// TwinCAT 3 PLC project Test
// ProgramVersion: 3.1.4024.0
// libraries:
//   Tc2_EtherCAT, * (Beckhoff Automation GmbH)
//   Tc2_Standard, * (Beckhoff Automation GmbH)
//   Tc2_System, * (Beckhoff Automation GmbH)
//   Tc3_Module, * (Beckhoff Automation GmbH)
// project tree:
//   DUTs/STRUCT/ Meca500SmPdo.TcDUT, SensorSmPdo.TcDUT
//   GVLs/ GVL.TcGVL
//   / PlcTask.TcTTO
//   POUs/ MAIN.TcPOU, Overall.TcPOU
// real-time tasks:
//   TASK PlcTask: cycle T#10ms, priority 20, ADS port 350
// I/O:
//   DEVICE Device 1 (EtherCAT), AmsNetId 192.168.0.153.2.1
//     Box 1 (Meca500) [Meca500]
//     Box 2 (Meca500) [Meca500]
//     Box 3 (BFT-MEDS-ECAT-M8) [BFT]
// variable links:
//   Test/Test Instance <-> Device 1 (EtherCAT)/Box 1 (Meca500)
//     PlcTask Inputs/GVL.Robot1.Inputs <-> SmPdoVariables/Meca500_SM_3
//     PlcTask Outputs/GVL.Robot1.Outputs <-> SmPdoVariables/Meca500_SM_2
//   Test/Test Instance <-> Device 1 (EtherCAT)/Box 2 (Meca500)
//     PlcTask Inputs/GVL.Robot2.Inputs <-> SmPdoVariables/Meca500_SM_3
//     PlcTask Outputs/GVL.Robot2.Outputs <-> SmPdoVariables/Meca500_SM_2
//   Test/Test Instance <-> Device 1 (EtherCAT)/Box 3 (BFT-MEDS-ECAT-M8)
//     PlcTask Inputs/GVL.Sensor.Inputs <-> SmPdoVariables/BFT_SM_3

CONFIGURATION Test
    RESOURCE PLC ON TwinCAT3
        TASK PlcTask(INTERVAL := T#10ms, PRIORITY := 20);
        PROGRAM MAIN WITH PlcTask : MAIN;
    END_RESOURCE
END_CONFIGURATION

// ---- DUTs/STRUCT/Meca500SmPdo.TcDUT
TYPE Meca500SmPdo :
STRUCT
	//From Ethercat Device SmPdos, Create this Structure by Enabling Create Sm/Pdo variable , in the Ethercat tab/Advance/Behavior
	Inputs 	AT %I* : ECAT_Meca500_SM_34A3A44A;	//for specific ESI firmware
	Outputs AT %Q* : ECAT_Meca500_SM_A587449F;	//for specific ESI firmware
	
	Connect					:	BOOL;	//Switch between Init State & OP State
	Connected				:	BOOL;	//Validate OP State
	DisconnectFromEthercat	:	BOOL;	//Send SDO command to disconnect from EtherCat and  switch to TCP
	ResettingPause			:	BOOL;	//Bit to indicate that cycling pause is in progress
	Ready					:	BOOL;	//Bit to indicate Robot is activated, homed, not in error and not in pause
	Stop					:	BOOL;	//Deactivate the robot motors

END_STRUCT
END_TYPE

// ---- DUTs/STRUCT/SensorSmPdo.TcDUT
TYPE SensorSmPdo :
STRUCT
	Inputs AT %I* : ECAT_BFT_SM_44E87B56;
	Outputs AT %Q* : ECAT_BFT_SM_911AEFB2;
END_STRUCT
END_TYPE

// ---- GVLs/GVL.TcGVL
{attribute 'qualified_only'}
VAR_GLOBAL
	Robot1	:	Meca500SmPdo;
	Robot2	:	Meca500SmPdo;
	Sensor :    SensorSmPdo;
	test:INT:=1;

END_VAR

// ---- POUs/MAIN.TcPOU
PROGRAM MAIN
VAR
	Values					:	ARRAY[1..11]OF REAL := [170,-30,150,0,90,0,2,32020,32021,0,0];	
	FirstScan				:	BOOL				:=  0;		
	StepSquareMove 			: 	INT 				:=  2;
	Select 					: 	INT 				:=  0;
	Overall 				: 	Overall;
	Error 					: 	BOOL 				:=  0;
	Sent 					: 	BOOL 				:=  0;
	Buffered 				: 	BOOL 				:=  0;	
	ExternalStatecontrol 	:	BOOL				:=  0;
	ExternalMove_ID			:	UINT				:=  0;	
END_VAR

Select := REAL_TO_INT(Values[11]);
StepSquareMove:=REAL_TO_INT(Values[10]);
//pos[1]:=GVL.Robot1.Inputs.End_Effector_Pose.SubIndex_001;
//pos[2]:=GVL.Robot1.Inputs.End_Effector_Pose.SubIndex_002;
//pos[3]:=GVL.Robot1.Inputs.End_Effector_Pose.SubIndex_003;
//pos[4]:=GVL.Robot1.Inputs.End_Effector_Pose.SubIndex_004;
//pos[5]:=GVL.Robot1.Inputs.End_Effector_Pose.SubIndex_005;
//pos[6]:=GVL.Robot1.Inputs.End_Effector_Pose.SubIndex_006;
			
//If ready to send move command
IF Select = 1 AND StepSquareMove = 1 THEN  // Robot1
	//send the appropriate values to move robot1
	//Joint_Angle: info for moving: this is an array of length 11 but only item 1-9 are used for movement			
	Overall(
			Joint_Angle:= Values, 
			ExternalStatecontrol:=0 , 
			ExternalMove_ID:=0 ,
			Robot:= GVL.Robot1 , 
			Error=> Error, 
			Sent:= Sent, 
			Buffered:= Buffered		
	);
	//If robot1 move is completed reset values
	IF Sent AND Buffered THEN
		Values[10]:=2;
		Sent:=0;
		Buffered:=0;
	END_IF 
	
ELSIF Select = 2 AND StepSquareMove = 1 THEN // Robot2
	//send the appropriate values to move robot2
	//Joint_Angle: info for moving: this is an array of length 11 but only item 1-9 are used for movement			
	Overall(
			Joint_Angle:= Values, 
			ExternalStatecontrol:=0 , 
			ExternalMove_ID:=0 ,
			Robot:= GVL.Robot2 , 
			Error=> Error, 
			Sent:= Sent, 
			Buffered:= Buffered		
	);
	//If robot2 move is completed reset values
	IF Sent AND Buffered THEN
		Values[10]:=2;
		Sent:=0;
		Buffered:=0;
	END_IF 
END_IF

END_PROGRAM

// ---- POUs/Overall.TcPOU
FUNCTION_BLOCK Overall
VAR_INPUT
	Joint_Angle				:	ARRAY[1..11]OF REAL;
	ExternalStatecontrol 	:	BOOL;
	ExternalMove_ID			:	UINT;
END_VAR
VAR_IN_OUT
	Robot	:	Meca500SmPdo;	
	Sent		:	BOOL;
	Buffered	:	BOOL;
END_VAR
VAR_OUTPUT
	Error		:	BOOL;
END_VAR
VAR
	Output_Params	:	ARRAY[1..6] OF REAL;
	FirstScan: BOOL:=0;
END_VAR

(*Collect Inputs and store them locally*)
Output_Params[1]:=Joint_Angle[1];
Output_Params[2]:=Joint_Angle[2];
Output_Params[3]:=Joint_Angle[3];
Output_Params[4]:=Joint_Angle[4];
Output_Params[5]:=Joint_Angle[5];
Output_Params[6]:=Joint_Angle[6];


(* If Values have change, Reinitialise Outputs*)

IF FirstScan=0 OR Robot.Outputs._Move.SubIndex_001 <> Output_Params[1] OR Robot.Outputs._Move.SubIndex_002 <> Output_Params[2] OR Robot.Outputs._Move.SubIndex_003 <> Output_Params[3] OR Robot.Outputs._Move.SubIndex_004 <> Output_Params[4] OR Robot.Outputs._Move.SubIndex_005 <> Output_Params[5] OR Robot.Outputs._Move.SubIndex_006 <> Output_Params[6] THEN
	Sent := FALSE;
	Buffered := FALSE;
END_IF;

(*if not in legacy mode, Activated Setpoint*)
IF Robot.Outputs.Motion_Control.Move_ID <> 0 THEN
    Robot.Outputs.Motion_Control.SetPoint := TRUE;
END_IF;

(* To send _Move, send _Move ID *)
IF NOT Buffered AND NOT Sent THEN
    
    Robot.Outputs._Move.Move_Command := REAL_TO_UDINT(Joint_Angle[7]);
    Robot.Outputs._Move.SubIndex_001 := Output_Params[1];
	Robot.Outputs._Move.SubIndex_002 := Output_Params[2];
	Robot.Outputs._Move.SubIndex_003 := Output_Params[3];
	Robot.Outputs._Move.SubIndex_004 := Output_Params[4];
	Robot.Outputs._Move.SubIndex_005 := Output_Params[5];
	Robot.Outputs._Move.SubIndex_006 := Output_Params[6];
	
    
    IF ExternalStateControl THEN
        IF ExternalMove_ID <> 0 AND ExternalMove_ID <> REAL_TO_UINT(Joint_Angle[8]) AND ExternalMove_ID <> REAL_TO_UINT(Joint_Angle[9]) THEN
            Robot.Outputs.Motion_Control.Move_ID := ExternalMove_ID;
            Sent := TRUE;
        END_IF;
        
    ELSE (*Not External Control*)
        IF Robot.Outputs.Motion_Control.Move_ID = REAL_TO_UINT(Joint_Angle[8]) THEN
            Robot.Outputs.Motion_Control.Move_ID := REAL_TO_UINT(Joint_Angle[9]);
        ELSIF Robot.Outputs.Motion_Control.Move_ID = REAL_TO_UINT(Joint_Angle[9]) THEN
            Robot.Outputs.Motion_Control.Move_ID := REAL_TO_UINT(Joint_Angle[8]);
        ELSIF Robot.Outputs.Motion_Control.Move_ID <> REAL_TO_UINT(Joint_Angle[8]) OR Robot.Outputs.Motion_Control.Move_ID <> REAL_TO_UINT(Joint_Angle[9]) THEN
            Robot.Outputs.Motion_Control.Move_ID := REAL_TO_UINT(Joint_Angle[8]);
        END_IF;
        Sent := TRUE;
    END_IF;
END_IF;

(* Check if _Move has been sent, if so, check if it was received *)
IF Sent THEN
    IF Robot.Outputs._Move.Move_Command = REAL_TO_UDINT(Joint_Angle[7]) THEN
        IF Robot.Outputs._Move.SubIndex_001 = Output_Params[1] AND Robot.Outputs._Move.SubIndex_002 = Output_Params[2] AND Robot.Outputs._Move.SubIndex_003 = Output_Params[3] AND Robot.Outputs._Move.SubIndex_004 = Output_Params[4] AND Robot.Outputs._Move.SubIndex_005 = Output_Params[5] AND Robot.Outputs._Move.SubIndex_006 = Output_Params[6] THEN
            IF Robot.Inputs.Motion_Status.Move_ID = Robot.Outputs.Motion_Control.Move_ID THEN
                Buffered := TRUE;
			//	Sent:=FALSE;
            END_IF;
        END_IF;
    END_IF;
END_IF;

(*If External _Move ID is equal to Internal, raise an error*)
IF ExternalMove_ID = REAL_TO_UINT(Joint_Angle[8]) OR ExternalMove_ID = REAL_TO_UINT(Joint_Angle[9]) THEN
    Error := TRUE;
END_IF;

FirstScan := TRUE;

END_FUNCTION_BLOCK
